TYPE CM_Motor_SIM :
STRUCT
END_STRUCT
END_TYPE

(* stored: Version 1.1.0.1, ProductVersion 3.1.4024.12
   DUT CM_Motor_SIM: Id {2d7575c0-ee7b-4702-adc0-a721667edef6} *)
